{attribute 'GeneratedUsingTerminal: EM7004-0000-0017'}
{attribute addProperty BoxType "EM7004-0000-0017"}
{attribute addProperty Id "Latch_extern_validBOOL1Set_counter_doneBOOL1Status_of_input_ABOOL1Status_of_input_BBOOL1Status_of_input_gateBOOL1Status_of_extern_latchBOOL1TxPDO_ToggleBOOL1"}
{attribute addProperty CRC "3027864966"}
{attribute addProperty Size "7"}
TYPE Status_B4798D86 :
STRUCT
	{attribute addProperty Name "Latch_extern_valid"}
	Latch_extern_valid : BOOL;
	{attribute addProperty Name "Set_counter_done"}
	Set_counter_done : BOOL;
	{attribute addProperty Name "Status_of_input_A"}
	Status_of_input_A : BOOL;
	{attribute addProperty Name "Status_of_input_B"}
	Status_of_input_B : BOOL;
	{attribute addProperty Name "Status_of_input_gate"}
	Status_of_input_gate : BOOL;
	{attribute addProperty Name "Status_of_extern_latch"}
	Status_of_extern_latch : BOOL;
	{attribute addProperty Name "TxPDO_Toggle"}
	TxPDO_Toggle : BOOL;
END_STRUCT
END_TYPE

(* stored: Version 1.2.0.0, ProductVersion 3.1.4024.9
   DUT Status_B4798D86: Id {be5e5236-0329-4504-95a1-e4ebab962e14} *)
